// TIA Portal project "profinets1" (V18)

(* hardware
DEVICE "S7-1200 station_1"  S7-1200 Station
   slot 0: "Rack_0"  S7-1200 Rack  Rack  V1.0
   slot 1: "PLC_1"  CPU 1214C AC/DC/Rly  6ES7 214-1BG40-0XB0  V4.1
   slot 2: "DI 8x24VDC/DQ 8xRelay_1"  SM 1223 DI8/DQ8 x relay  6ES7 223-1PH32-0XB0  V2.0
   slot 3: "AQ 2x14BIT_1"  SM 1232 AQ2  6ES7 232-4HB32-0XB0  V2.1
   slot 101: "CM 1241 (RS422/485)_1"  6ES7 241-1CH32-0XB0  V2.2
DEVICE "GSD device_1"  GSD.Device.PN
   slot 0: "机架"  Rack  V1.0
   slot 0: "pn248"  BASIC V1.2  0  V1.2
      slot 0: "Robot Basic Device"  Robot Basic Device  0  V1.2
      slot 1: "PROFINET Interface"  PROFINET Interface
         slot 1: "Network Port"  Network Port
   slot 1: "DI 64 bytes_1"  DI 64 bytes
      slot 0: "DI 64 bytes"  DI 64 bytes
   slot 2: "DO 64 bytes_1"  DO 64 bytes
      slot 0: "DO 64 bytes"  DO 64 bytes
*)

// ===== PLC "PLC_1"  CPU 1214C AC/DC/Rly =====

VAR_GLOBAL   // PLC tag table "默认变量表"
   "Tag_1" AT %IB68 : Byte;
   "Tag_2" AT %MB10 : Byte;
   "Tag_3" AT %MB20 : Byte;
   "Tag_4" AT %QB68 : Byte;
   "PN_GO_8_15" AT %IB69 : Byte;
   "PN_GI_8_15" AT %QB69 : Byte;
   "Tag_7" AT %MB21 : Byte;
   "Tag_8" AT %MB11 : Byte;
   "Tag_9" AT %Q0.1 : Bool;
   "Tag_10" AT %Q0.6 : Bool;
   "PN_DI_0" AT %Q68.0 : Bool;
   "Tag_12" AT %Q0.4 : Bool;
   "Tag_13" AT %Q0.5 : Bool;
   "Tag_14" AT %Q0.7 : Bool;
   "Tag_15" AT %Q0.0 : Bool;
   "PN_DO_0" AT %I68.0 : Bool;
   "Tag_17" AT %M0.1 : Bool;
   "Tag_18" AT %M1.1 : Bool;
   "Tag_19" AT %M0.0 : Bool;
   "Tag_20" AT %M1.0 : Bool;
   "Tag_21" AT %QB32 : Byte;
   "Tag_5" AT %MB69 : Byte;
   "Tag_6" AT %QB0 : Byte;
   "Tag_11" AT %MB68 : Byte;
   "Tag_16" AT %I0.0 : Bool;
   "Tag_22" AT %I0.1 : Bool;
   "Tag_23" AT %I0.7 : Bool;
   "Tag_24" AT %M50.0 : Bool;
   "Tag_25" AT %M70.0 : Bool;
   "Tag_26" AT %M80.0 : Bool;
   "Tag_27" AT %I80.0 : Bool;
   "Tag_28" AT %Q90.0 : Bool;
   "Tag_29" AT %M70.1 : Bool;
   "Tag_30" AT %Q68.1 : Bool;
   "Tag_31" AT %M70.2 : Bool;
   "Tag_32" AT %Q68.2 : Bool;
   "Tag_33" AT %Q0.2 : Bool;
   "Tag_34" AT %M70.7 : Bool;
   "Tag_35" AT %MB70 : Byte;
   "Tag_36" AT %M70.3 : Bool;
   "Tag_37" AT %Q68.3 : Bool;
   "Tag_38" AT %Q0.3 : Bool;
   "Tag_39" AT %M70.4 : Bool;
   "Tag_40" AT %Q68.4 : Bool;
END_VAR

ORGANIZATION_BLOCK "Main"   // OB1, LAD, ProgramCycle
TITLE = "Main Program Sweep (Cycle)"
{ S7_Optimized_Access := 'TRUE' }
VERSION : 0.1
   VAR_INPUT
      Initial_Call : Bool;   // Initial call of this OB
      Remanence : Bool;   // =True, if remanent data are available
   END_VAR
BEGIN

REGION Network 1
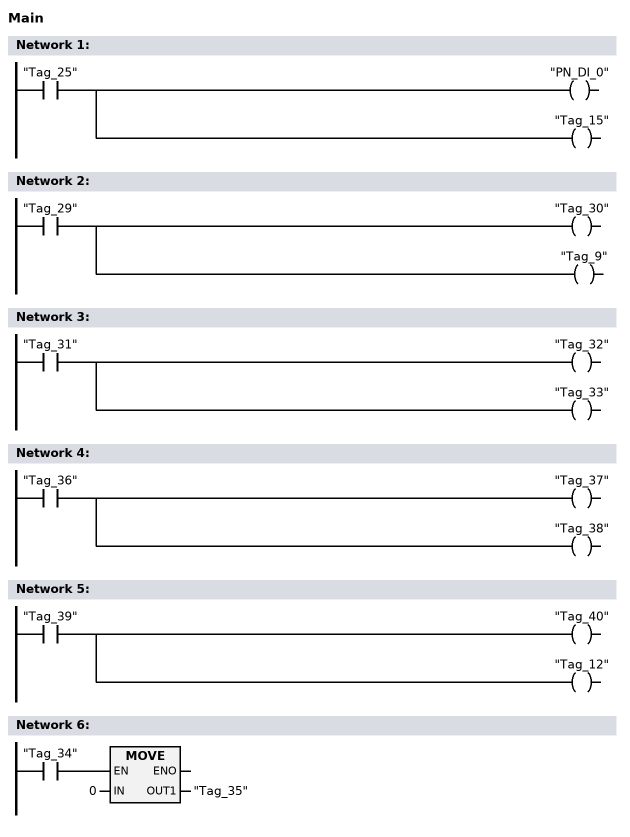
   RUNG wire#powerrail
      Contact( "Tag_25" )
      wire#w1
      Coil( "PN_DI_0" )
   END_RUNG
   RUNG wire#w1
      Coil( "Tag_15" )
   END_RUNG
   // the same network as SCL:
   "PN_DI_0" := "Tag_25";
   "Tag_15" := "Tag_25";
END_REGION

REGION Network 2
   RUNG wire#powerrail
      Contact( "Tag_29" )
      wire#w1
      Coil( "Tag_30" )
   END_RUNG
   RUNG wire#w1
      Coil( "Tag_9" )
   END_RUNG
   // the same network as SCL:
   "Tag_30" := "Tag_29";
   "Tag_9" := "Tag_29";
END_REGION

REGION Network 3
   RUNG wire#powerrail
      Contact( "Tag_31" )
      wire#w1
      Coil( "Tag_32" )
   END_RUNG
   RUNG wire#w1
      Coil( "Tag_33" )
   END_RUNG
   // the same network as SCL:
   "Tag_32" := "Tag_31";
   "Tag_33" := "Tag_31";
END_REGION

REGION Network 4
   RUNG wire#powerrail
      Contact( "Tag_36" )
      wire#w1
      Coil( "Tag_37" )
   END_RUNG
   RUNG wire#w1
      Coil( "Tag_38" )
   END_RUNG
   // the same network as SCL:
   "Tag_37" := "Tag_36";
   "Tag_38" := "Tag_36";
END_REGION

REGION Network 5
   RUNG wire#powerrail
      Contact( "Tag_39" )
      wire#w1
      Coil( "Tag_40" )
   END_RUNG
   RUNG wire#w1
      Coil( "Tag_12" )
   END_RUNG
   // the same network as SCL:
   "Tag_40" := "Tag_39";
   "Tag_12" := "Tag_39";
END_REGION

REGION Network 6
   RUNG wire#powerrail
      Contact( "Tag_34" )
      Move(in := 0, out1 => "Tag_35")
   END_RUNG
   // the same network as SCL:
   IF "Tag_34" THEN "Tag_35" := 0; END_IF;
END_REGION
END_ORGANIZATION_BLOCK